// TIA Portal V19 export
FUNCTION_BLOCK "Main_Safety_RTG1"   // FB, F_LAD
{ S7_Optimized_Access := 'TRUE' }
// stored: AutoNumber false
BEGIN

REGION Network 1
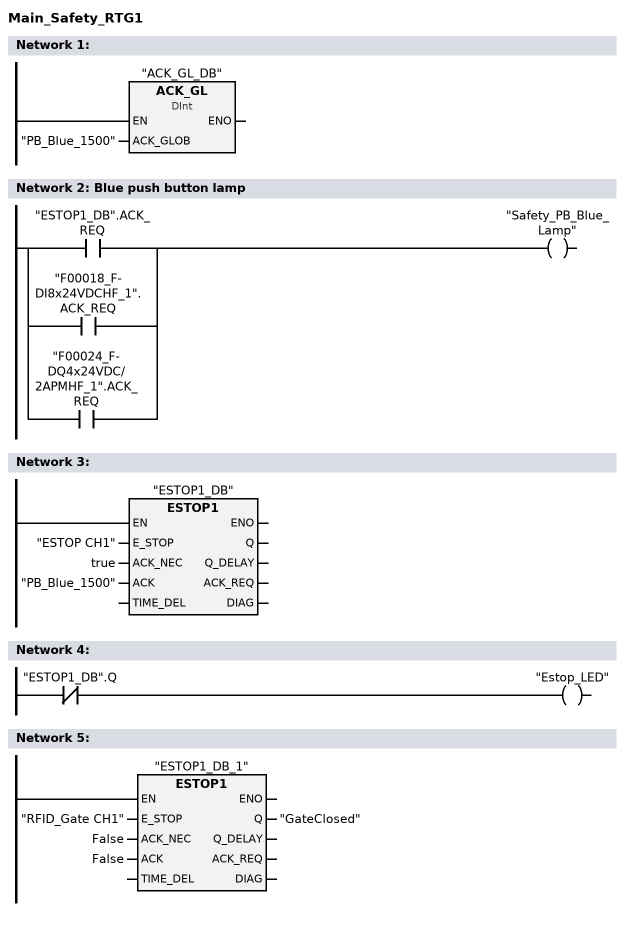
   RUNG wire#powerrail
      { S7_Templates := "codedbool_type := DInt" } "ACK_GL_DB".ACK_GL(ACK_GLOB := "PB_Blue_1500")
   END_RUNG
   // the same network as SCL:
   "ACK_GL_DB"(ACK_GLOB := "PB_Blue_1500");   // ACK_GL
END_REGION

REGION Network 2: Blue push button lamp
   RUNG wire#powerrail
      Contact( "ESTOP1_DB".ACK_REQ )
      wire#w1
      Coil( "Safety_PB_Blue_Lamp" )
   END_RUNG
   RUNG wire#powerrail
      Contact( "F00018_F-DI8x24VDCHF_1".ACK_REQ )
   END_RUNG wire#w1
   RUNG wire#powerrail
      Contact( "F00024_F-DQ4x24VDC/2APMHF_1".ACK_REQ )
   END_RUNG wire#w1
   // the same network as SCL:
   "Safety_PB_Blue_Lamp" := "ESTOP1_DB".ACK_REQ OR "F00018_F-DI8x24VDCHF_1".ACK_REQ OR "F00024_F-DQ4x24VDC/2APMHF_1".ACK_REQ;
END_REGION

REGION Network 3
   RUNG wire#powerrail
      "ESTOP1_DB".ESTOP1(E_STOP := "ESTOP CH1", ACK_NEC := true, ACK := "PB_Blue_1500", TIME_DEL :=, Q =>, Q_DELAY =>, ACK_REQ =>, DIAG =>)
   END_RUNG
   // the same network as SCL:
   "ESTOP1_DB"(E_STOP := "ESTOP CH1", ACK_NEC := true, ACK := "PB_Blue_1500");   // ESTOP1
END_REGION

REGION Network 4
   RUNG wire#powerrail
      I_Contact( "ESTOP1_DB".Q )
      Coil( "Estop_LED" )
   END_RUNG
   // the same network as SCL:
   "Estop_LED" := NOT "ESTOP1_DB".Q;
END_REGION

REGION Network 5
   RUNG wire#powerrail
      "ESTOP1_DB_1".ESTOP1(E_STOP := "RFID_Gate CH1", ACK_NEC := False, ACK := False, TIME_DEL :=, Q => "GateClosed", Q_DELAY =>, ACK_REQ =>, DIAG =>)
   END_RUNG
   // the same network as SCL:
   "ESTOP1_DB_1"(E_STOP := "RFID_Gate CH1", ACK_NEC := False, ACK := False, Q => "GateClosed");   // ESTOP1
END_REGION
END_FUNCTION_BLOCK
